FUNCTION_BLOCK Section3Ctrl (* Basic Function Block Type *)
  (* Standard: 61499-2 *)
  (* Version 0.0, 5/27/2018, MIA, nxtControl GmbH, Template *)
  PACKAGE Main;
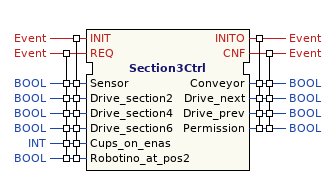
  EVENT_INPUT
    INIT WITH Sensor, Drive_section2, Drive_section4, Drive_section6, Cups_on_enas, Robotino_at_pos2; (* Initialization Request *)
    REQ WITH Sensor, Drive_section2, Drive_section4, Drive_section6, Cups_on_enas, Robotino_at_pos2; (* Normal Execution Request *)
  END_EVENT
  EVENT_OUTPUT
    INITO WITH Conveyor, Drive_next, Drive_prev, Permission; (* Initialization Confirm *)
    CNF WITH Conveyor, Drive_next, Drive_prev, Permission; (* Execution Confirmation *)
  END_EVENT
  VAR_INPUT
    Sensor : BOOL; (* Input event qualifier *)
    Drive_section2 : BOOL;
    Drive_section4 : BOOL;
    Drive_section6 : BOOL;
    Cups_on_enas : INT;
    Robotino_at_pos2 : BOOL;
  END_VAR
  VAR_OUTPUT
    Conveyor : BOOL; (* Output event qualifier *)
    Drive_next : BOOL;
    Drive_prev : BOOL;
    Permission : BOOL;
  END_VAR
  VAR
    TimeStamp : DATE_AND_TIME;
  END_VAR
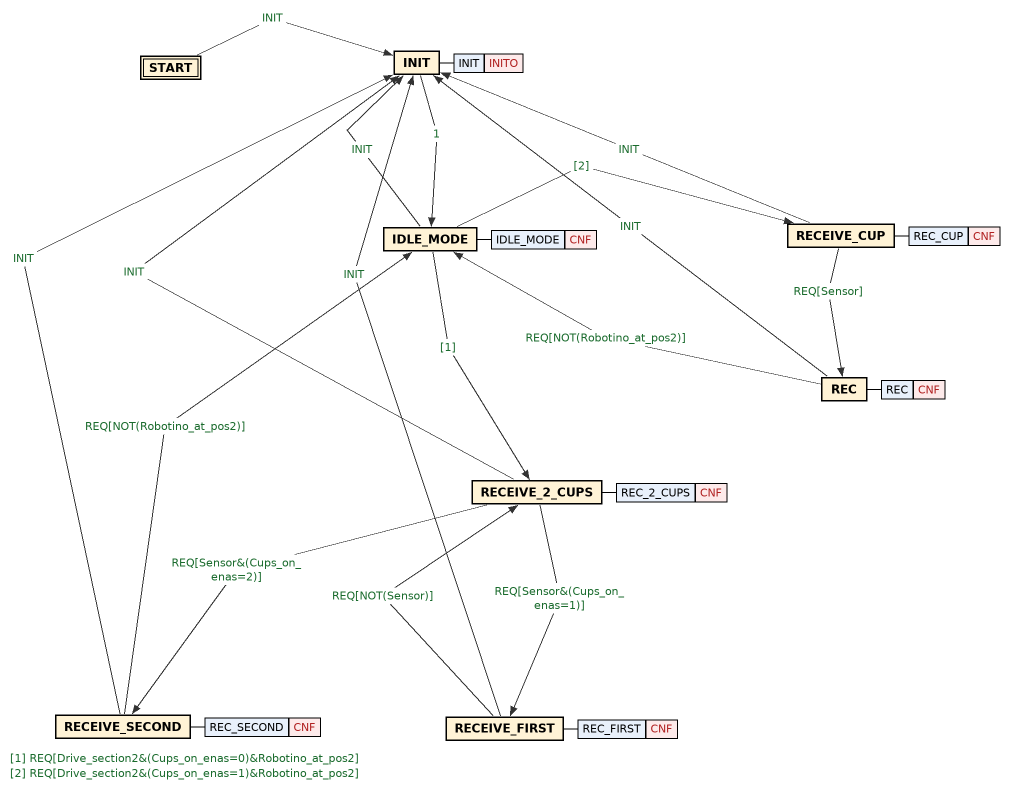
  EC_STATES
    START; (* Initial State *)
    INIT : INIT -> INITO; (* Initialization *)
    IDLE_MODE : IDLE_MODE -> CNF;
    RECEIVE_2_CUPS : REC_2_CUPS -> CNF;
    RECEIVE_FIRST : REC_FIRST -> CNF;
    RECEIVE_SECOND : REC_SECOND -> CNF;
    RECEIVE_CUP : REC_CUP -> CNF;
    REC : REC -> CNF;
  END_STATES
  EC_TRANSITIONS
    START TO INIT := INIT;
    INIT TO IDLE_MODE := 1;
    IDLE_MODE TO INIT := INIT;
    IDLE_MODE TO RECEIVE_2_CUPS := REQ[Drive_section2&(Cups_on_enas=0)&Robotino_at_pos2];
    RECEIVE_2_CUPS TO RECEIVE_FIRST := REQ[Sensor&(Cups_on_enas=1)];
    RECEIVE_FIRST TO RECEIVE_2_CUPS := REQ[NOT(Sensor)];
    RECEIVE_2_CUPS TO RECEIVE_SECOND := REQ[Sensor&(Cups_on_enas=2)];
    RECEIVE_SECOND TO IDLE_MODE := REQ[NOT(Robotino_at_pos2)];
    IDLE_MODE TO RECEIVE_CUP := REQ[Drive_section2&(Cups_on_enas=1)&Robotino_at_pos2];
    RECEIVE_CUP TO REC := REQ[Sensor];
    REC TO IDLE_MODE := REQ[NOT(Robotino_at_pos2)];
    RECEIVE_CUP TO INIT := INIT;
    REC TO INIT := INIT;
    RECEIVE_SECOND TO INIT := INIT;
    RECEIVE_2_CUPS TO INIT := INIT;
    RECEIVE_FIRST TO INIT := INIT;
  END_TRANSITIONS
  ALGORITHM INIT IN ST: (* Initialization algorithm *)
Conveyor := FALSE;
Drive_prev := FALSE;
Drive_next := FALSE;
Permission := FALSE;
  END_ALGORITHM
  ALGORITHM IDLE_MODE IN ST:
Conveyor := FALSE;
Drive_prev := TRUE;
Drive_next := FALSE;
Permission := FALSE;
  END_ALGORITHM
  ALGORITHM REC_2_CUPS IN ST:
Conveyor := TRUE;
Drive_prev := TRUE;
Drive_next := FALSE;
Permission := FALSE;
  END_ALGORITHM
  ALGORITHM REC_FIRST IN ST:
Conveyor := TRUE;
Drive_prev := TRUE;
Drive_next := TRUE;
Permission := TRUE;
  END_ALGORITHM
  ALGORITHM REC_SECOND IN ST:
Conveyor := FALSE;
Drive_prev := FALSE;
Drive_next := FALSE;
Permission := TRUE;
  END_ALGORITHM
  ALGORITHM REC_CUP IN ST:
Conveyor := TRUE;
Drive_prev := TRUE;
Drive_next := TRUE;
Permission := FALSE;
  END_ALGORITHM
  ALGORITHM REC IN ST:
Conveyor := FALSE;
Drive_prev := FALSE;
Drive_next := FALSE;
Permission := TRUE;
  END_ALGORITHM
END_FUNCTION_BLOCK
